// TwinCAT 3 PLC project ControlControls
// ProgramVersion: 3.1.4024.0
// libraries:
//   Tc2_Standard, * (Beckhoff Automation GmbH)
//   Tc2_System, * (Beckhoff Automation GmbH)
//   Tc3_Module, * (Beckhoff Automation GmbH)
//   VisuSymbols,3.5.10.0,System
// project tree:
//   / GlobalTextList.TcGTLO, PlcTask.TcTTO, Visualization Manager.TcVMO (not stored), VISU_TASK.TcTTO
//   GVLs/ GVL.TcGVL
//   POUs/ MAIN.TcPOU
//   VISUs/ Visualization.TcVIS
// real-time tasks:
//   TASK PlcTask: cycle T#10ms, priority 20, ADS port 350
//   TASK VISU_TASK: cycle T#200000us, priority 30, ADS port 351
// I/O:
//   DEVICE Device 1 (EtherCAT), AmsNetId 199.4.42.250.2.1
//     Term 1 (EK1100) [EK1100 EtherCAT Coupler (2A E-Bus)]
//       Term 2 (EL1008) [EL1008 8Ch. Dig. Input 24V, 3ms]
//       Term 3 (EL1008) [EL1008 8Ch. Dig. Input 24V, 3ms]
//       Term 4 (EL2008) [EL2008 8Ch. Dig. Output 24V, 0.5A]
//       Term 5 (EL2008) [EL2008 8Ch. Dig. Output 24V, 0.5A]
//       Term 6 (EL3002) [EL3002 2Ch. Ana. Input +/-10V]
//       Term 7 (EL4002) [EL4002 2Ch. Ana. Output 0-10V, 12bit]
//       Term 8 (EL3124) [EL3124 4Ch. Ana. Input 4-20mA Diff.]
//       Term 9 (EL4024) [EL4024 4Ch. Ana. Output 4-20mA, 12bit]
//       Box 10 (BK1250)
//     Term 11 (EK1100) [EK1100 EtherCAT Coupler (2A E-Bus)]
//       Term 12 (EL1008) [EL1008 8Ch. Dig. Input 24V, 3ms]
//       Term 13 (EL2008) [EL2008 8Ch. Dig. Output 24V, 0.5A]
//       Term 14 (EL9011) [EL9011 End Terminal]
// variable links:
//   ControlControls/ControlControls Instance <-> Device 1 (EtherCAT)/Term 11 (EK1100)/Term 12 (EL1008)
//     PlcTask Inputs/GVL.bS{1..5} <-> Channel {1..5}/GVL.bS{1..5}  (5 links)
//     PlcTask Inputs/GVL.bStart_B1 <-> Channel 6/GVL.bStart_B1
//     PlcTask Inputs/GVL.bStop_B2 <-> Channel 7/GVL.bStop_B2
//   ControlControls/ControlControls Instance <-> Device 1 (EtherCAT)/Term 11 (EK1100)/Term 13 (EL2008)
//     PlcTask Outputs/GVL.LightOn <-> Channel 6/GVL.LightOn
//     PlcTask Outputs/GVL.bA1 <-> Channel 2/GVL.bA1
//     PlcTask Outputs/GVL.bA2 <-> Channel 3/GVL.bA2
//     PlcTask Outputs/GVL.bA3 <-> Channel 5/GVL.bA3
//     PlcTask Outputs/GVL.bMotor_M1 <-> Channel 1/GVL.bMotor_M1
//     PlcTask Outputs/GVL.bMotor_M2 <-> Channel 4/GVL.bMotor_M2

CONFIGURATION ControlControls
    RESOURCE PLC ON TwinCAT3
        TASK PlcTask(INTERVAL := T#10ms, PRIORITY := 20);
        TASK VISU_TASK(INTERVAL := T#200000us, PRIORITY := 30);
        PROGRAM MAIN WITH PlcTask : MAIN;
        PROGRAM VisuElems_Visu_Prg WITH VISU_TASK : VisuElems.Visu_Prg;
    END_RESOURCE
END_CONFIGURATION

// ---- GVLs/GVL.TcGVL
{attribute 'qualified_only'}
VAR_GLOBAL
		//Input
	bS1 AT %I*: BOOL;
	bS2 AT %I*: BOOL;
	bS3 AT %I*: BOOL;
	bS4 AT %I*: BOOL;
	bS5 AT %I*: BOOL;
	
	bStart_B1 AT %I* : BOOL;
	bStop_B2 AT %I* : BOOL;
	
	start: BOOL;
	stop:BOOL;
	
	//output
	bMotor_M1 AT %Q* : BOOL;
	bMotor_M2 AT %Q* : BOOL;
	bA1 AT %Q* : BOOL;
	bA2 AT %Q* : BOOL;
	bA3 AT %Q* : BOOL;
	LightOn AT %Q* : BOOL;
	
	
	
	bA1PLACTIC_COUNT: INT;
	CD: INT;
	LOAD: INT;
	PV: INT;
	Q: INT;
	CV: INT;
END_VAR

// ---- POUs/MAIN.TcPOU
PROGRAM MAIN
VAR
	
	TimerP01: TON;
	Timer02: TON;
	
	MotorActive: BOOL;
	P_COUNT: INT:=0;
	P_LIMIT: INT:=3;
	
	M_COUNT:INT:=0;
	M_LIMIT: INT:=3;
	
	Wastage: INT:=0;
	FinalProduct: INT:=0;
	
	bS1Detect: BOOL;
	bS2Detect: BOOL; 
	bs3Detect: BOOL;
	bs4Detect: BOOL; 
	bs5Detect: BOOL;
	
	tTimer01: TOF;
	timerReset: RS;
	bs1triger: R_TRIG;
	bs4Triger: R_TRIG;
	bs5Triger: F_TRIG;
	bs2Triger: R_TRIG;
	
	
	bs5RTriger: R_TRIG;
	
	bA2Timer: TON;
	
	bA2OpenTime: TON;
	bA1PopTimer: TON;
	bs3triger: R_TRIG;
	fbTimerOn: TON;
	fbTimerOff: TOF;
	
	timerOnRunning: BOOL:=FALSE;
	
	
	
	lightOnTimer: TOF;
	bA3PopTime: TON;
	bs5RDetect: BOOL;
	Plactic_Count: INT;
	MetalCount: INT;
END_VAR

//......................................Motor Control........................................

//Start the motor
IF GVL.bStart_B1 OR GVL.start THEN
    MotorActive:=TRUE;	
END_IF

IF MotorActive THEN
	GVL.bMotor_M1:=TRUE;
	GVL.bMotor_M2:=TRUE;
END_IF

//Stop the motor
IF GVL.bStop_B2 OR GVL.STOP THEN
    GVL.bMotor_M1 := FALSE;
    GVL.bMotor_M2 := FALSE;
	MotorActive:=FALSE;
END_IF;

//......................................Edge Detection........................................

//bs1 rising edge detection
bs1triger(CLK:=GVL.bS1);
IF bs1triger.Q THEN
	bs1Detect:= TRUE;	
END_IF

//bs2 rising edge detection 
bs2Triger(CLK:=GVL.bS2);
IF bs2Triger.Q THEN	
	bs2Detect:=TRUE;
END_IF
//bs3 rising edge detection
bs3triger(CLK:=GVL.bS3);
IF bs3Triger.Q THEN
	bs3Detect:=TRUE;
END_IF

//bs4 Rising edge detection
bs4Triger(CLK:=GVL.bS4 );
IF bs4Triger.Q THEN
	bs4Detect:=TRUE;	
END_IF
//bs5 Rising edge detection
bs5RTriger(CLK:=GVL.bS4);
IF bs5RTriger.Q THEN
	bs5RDetect:=TRUE;	
END_IF

//bs5 Falling edge detection
bs5Triger(CLK:=GVL.bS5);
IF bs5Triger.Q THEN
	bs5Detect:=TRUE;
END_IF

//.....................................Plastic Sortor Control....................................

//bs1 sensor detection and bA1 solenoid Activation
IF bs1Detect and NOT(bs2Detect)THEN
	
	IF P_COUNT < P_LIMIT THEN
		//tTimer01(IN:=bs1Detect AND NOT(GVL.bS2),PT:= T#100MS , Q=> , ET=> );
	
		TimerP01(IN:=TRUE , PT:= T#800mS, );
		IF TimerP01.Q THEN
			
			//IF GVL.bA1=FALSE THEN
				GVL.bA1:=TRUE;
				bA1PopTimer(IN:=TRUE, PT:=T#100MS );
				
				IF bA1PopTimer.Q THEN
					GVL.bA1:=FALSE;
					P_COUNT := P_COUNT+1;
					bs1Detect:=FALSE;
					
				END_IF
			
		END_IF
		
	ELSE		
		GVL.bA1:=FALSE;	
	END_IF 
ELSE
	TimerP01(IN := FALSE);
    bA1PopTimer(IN := FALSE);
	//tTimer01(IN := FALSE);	
END_IF
IF P_COUNT>0 THEN
	Plactic_Count:=P_COUNT;
END_IF



//............................................Metal Sortor Control........................................

// Counting and bA2 solenoid activation
IF M_COUNT < M_LIMIT THEN	
	IF bs2Detect AND bs1Detect THEN
		bA2Timer(IN:=TRUE, PT:=T#1S );
		IF bA2Timer.Q THEN
			//IF GVL.bA2=FALSE THEN
				GVL.bA2:=TRUE;
				
				bA2OpenTime(IN:=TRUE , PT:=T#1S);
				
				IF bA2OpenTime.Q THEN
					GVL.bA2:=FALSE;
					M_COUNT:=M_COUNT+1;
					
					bs2Detect:=FALSE;
				END_IF

		END_IF
	
	ELSE
		
		bA2Timer(IN:=FALSE);
		bA2OpenTime(IN:=FALSE);
	END_IF
ELSE 
	M_COUNT:=0;
	
END_IF
IF M_COUNT>0 THEN
	MetalCount:=M_COUNT;
	
END_IF


// the plastic count -
IF bs2Detect THEN
	IF P_COUNT > 0 THEN
		P_COUNT := P_COUNT - 1;
	END_IF
END_IF


//......................................Wastage Management...................................................

IF bs4Detect THEN
    
    IF  bs5Detect  THEN
        GVL.bA3 := FALSE;   
        FinalProduct:=FinalProduct+1;
        bs4Detect := FALSE; 
        bs5Detect := FALSE; 
    ELSE
        
        Timer02(IN := TRUE, PT := T#600MS);  
        IF Timer02.Q THEN
            GVL.bA3 := TRUE; 
            bA3PopTime(IN := TRUE, PT := T#100MS);  
            
            IF bA3PopTime.Q THEN
                GVL.bA3 := FALSE;  
                Wastage := Wastage + 1;  
                bs4Detect := FALSE; 
            END_IF
        END_IF
    END_IF
ELSE
   
    GVL.bA3 := FALSE;
    Timer02(IN := FALSE);
    bA3PopTime(IN := FALSE);
END_IF


//..................................Blinking the light when wastage is detected................................

fbTimerOff(IN:=bs4Detect AND bs5RDetect,PT:=T#2S);
IF fbTimerOff.Q THEN
	timerOnRunning:= NOT timerOnRunning;
		//fbTimerOff(IN:=FALSE);
ELSE
	GVL.LightOn:=FALSE;
	fbTimerOff(IN:=False);
				
END_IF
	GVL.LightOn:=timerOnRunning;
	

//LIGHT ON (FINAL PRODUCT INDICATION)
lightOnTimer(IN:=bs5RDetect , PT:=T#2S);
IF lightOnTimer.Q THEN	
		timerOnRunning:=TRUE;
ELSE
	GVL.LightOn:=FALSE;
	lightOnTimer(IN:=FALSE);
END_IF
GVL.LightOn:=timerOnRunning;

END_PROGRAM

// ---- GlobalTextList.TcGTLO
TEXTLIST GlobalTextList
  866 = '%d'
  582 = '%S'
  130 = '%s'
  826 = 'COUNTING'
  806 = 'kk'
  182 = 'metal'
  184 = 'METAL'
  328 = 'Motor Control'
  9 = 'PLACTIC'
  702 = 'plactic Count'
  613 = 'PLASCTIC'
  569 = 'PLASCTIC STANDBY'
  385 = 'PLASTIC STANDBY'
  783 = 'PRODUCT'
  769 = 'START'
  659 = 'STOP'
  371 = 'WASTAGE'
END_TEXTLIST

// ---- VISUs/Visualization.TcVIS
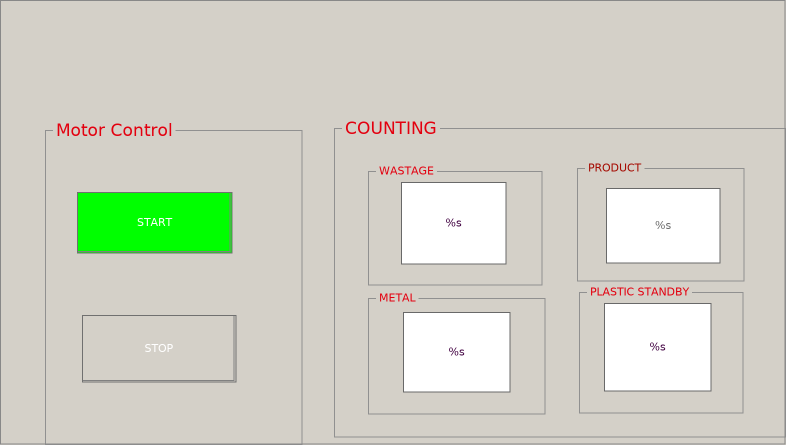
VISUALIZATION Visualization  // 786x445
    GroupBox (45,122 257x323), "Motor Control"
        Button (32,70 155x61), "START", text variable: GVL.start
        Button (37,193 154x67), "STOP", text variable: GVL.stop
    GroupBox (334,120 452x317), "COUNTING"
        GroupBox (34,43 174x122), "WASTAGE"
            Textfield (33,19 105x82), "%s", text variable: MAIN.Wastage
        GroupBox (243,40 167x121), "PRODUCT"
            Textfield (29,28 114x75), "%s", text variable: MAIN.FinalProduct
        GroupBox (34,170 177x124), "METAL"
            Textfield (35,22 107x80), "%s", text variable: MAIN.MetalCount
        GroupBox (245,164 164x129), "PLASTIC STANDBY"
            Textfield (25,19 107x88), "%s", text variable: MAIN.Plactic_Count
END_VISUALIZATION
